Yaskawa INFORM job: PSTART-SAMPLE.JBI

/JOB
//NAME PSTART-SAMPLE
//POS
///NPOS 0,0,0,0,0,0
//INST
///DATE 2023/02/06 16:47
///ATTR SC,RW,CJ
NOP
PSTART JOB:R1-MOVE SUB1
PSTART JOB:R2-MOVE SUB2
PSTART JOB:S1-MOV SUB3
PWAIT SUB1
PWAIT SUB2
PWAIT SUB3
END
